TYPE UDT_SensorInput :
STRUCT
	Link: BOOL;
	FilterTime: DINT;
END_STRUCT
END_TYPE

(* stored: Version 1.1.0.1, ProductVersion 3.1.4022.16
   DUT UDT_SensorInput: Id {a61dbd50-50d8-495b-89eb-257083d62514} *)
